PROGRAM Stn6
VAR

	start6: BOOL;
	reset6: BOOL;

	Stn6ProcessFE: F_TRIG;
	Stn6ProcessRE: R_TRIG;
	bCutStn6ProcessHalt: BOOL;
	DoorClose6: R_TRIG;
	bStn6DoorClamp: BOOL;

END_VAR
VAR // added by the converter: edge detectors and wires of the graphical bodies
    _w1, _w2 : ANY;
    _w3 : BOOL;
END_VAR

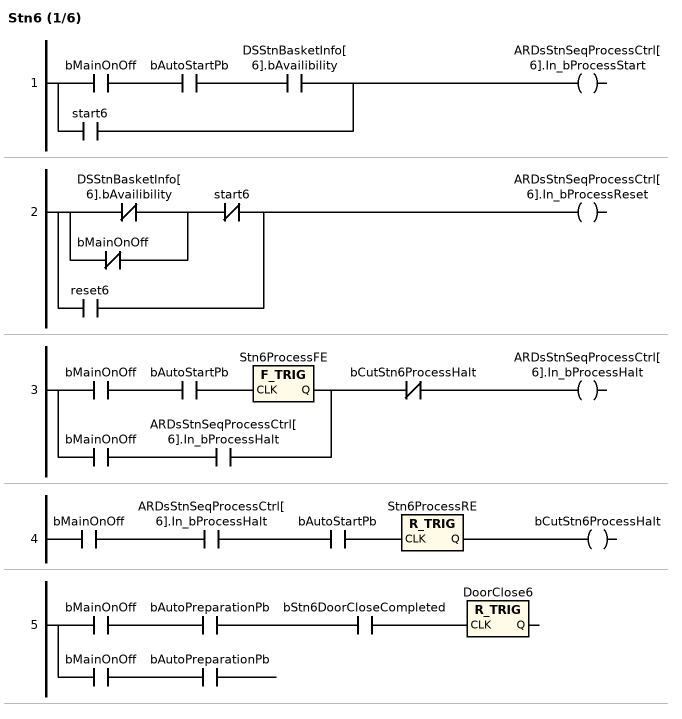
// NETWORK 1
ARDsStnSeqProcessCtrl[6].In_bProcessStart := bMainOnOff AND bAutoStartPb AND DSStnBasketInfo[6].bAvailibility OR start6;

// NETWORK 2
ARDsStnSeqProcessCtrl[6].In_bProcessReset := (NOT DSStnBasketInfo[6].bAvailibility OR NOT bMainOnOff) AND NOT start6 OR reset6;

// NETWORK 3
Stn6ProcessFE(CLK := bMainOnOff AND bAutoStartPb); // F_TRIG
ARDsStnSeqProcessCtrl[6].In_bProcessHalt := (Stn6ProcessFE.Q OR bMainOnOff AND ARDsStnSeqProcessCtrl[6].In_bProcessHalt) AND NOT bCutStn6ProcessHalt;

// NETWORK 4
Stn6ProcessRE(CLK := bMainOnOff AND ARDsStnSeqProcessCtrl[6].In_bProcessHalt AND bAutoStartPb); // R_TRIG
bCutStn6ProcessHalt := Stn6ProcessRE.Q;

// NETWORK 5
DoorClose6(CLK := bMainOnOff AND bAutoPreparationPb AND bStn6DoorCloseCompleted); // R_TRIG
(* DoorClose6.Q OR bMainOnOff AND bAutoPreparationPb; result not used *)

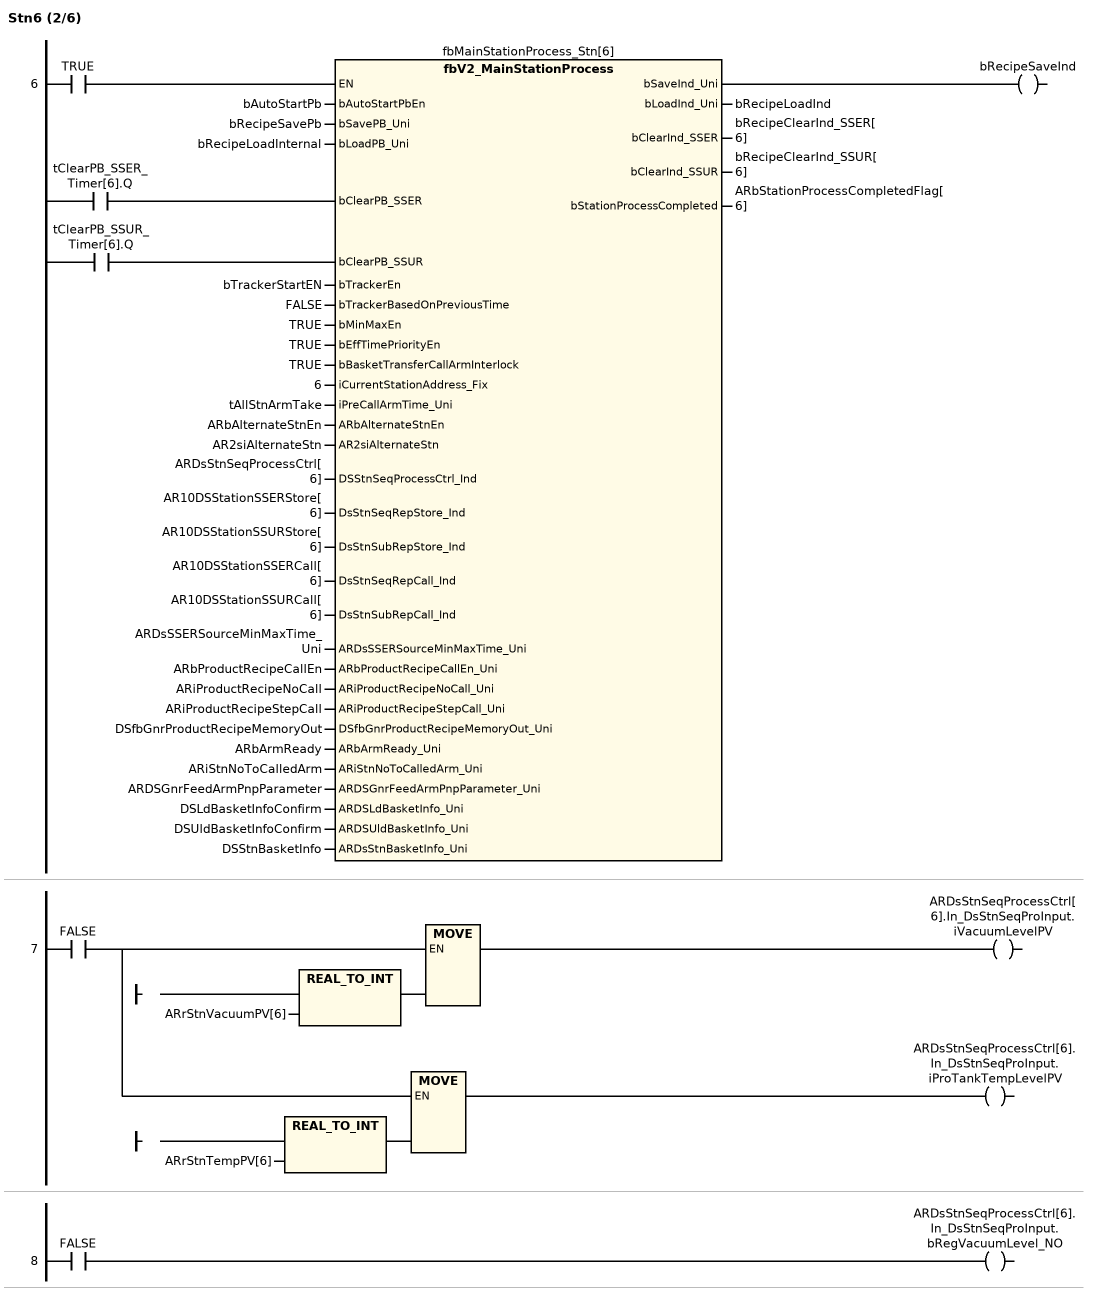
// NETWORK 6
fbMainStationProcess_Stn[6](
    bAutoStartPbEn := bAutoStartPb,
    bSavePB_Uni := bRecipeSavePb,
    bLoadPB_Uni := bRecipeLoadInternal,
    bClearPB_SSER := tClearPB_SSER_Timer[6].Q,
    bClearPB_SSUR := tClearPB_SSUR_Timer[6].Q,
    bTrackerEn := bTrackerStartEN,
    bTrackerBasedOnPreviousTime := FALSE,
    bMinMaxEn := TRUE,
    bEffTimePriorityEn := TRUE,
    bBasketTransferCallArmInterlock := TRUE,
    iCurrentStationAddress_Fix := 6,
    iPreCallArmTime_Uni := tAllStnArmTake,
    ARbAlternateStnEn := ARbAlternateStnEn,
    AR2siAlternateStn := AR2siAlternateStn,
    DSStnSeqProcessCtrl_Ind := ARDsStnSeqProcessCtrl[6],
    DsStnSeqRepStore_Ind := AR10DSStationSSERStore[6],
    DsStnSubRepStore_Ind := AR10DSStationSSURStore[6],
    DsStnSeqRepCall_Ind := AR10DSStationSSERCall[6],
    DsStnSubRepCall_Ind := AR10DSStationSSURCall[6],
    ARDsSSERSourceMinMaxTime_Uni := ARDsSSERSourceMinMaxTime_Uni,
    ARbProductRecipeCallEn_Uni := ARbProductRecipeCallEn,
    ARiProductRecipeNoCall_Uni := ARiProductRecipeNoCall,
    ARiProductRecipeStepCall_Uni := ARiProductRecipeStepCall,
    DSfbGnrProductRecipeMemoryOut_Uni := DSfbGnrProductRecipeMemoryOut,
    ARbArmReady_Uni := ARbArmReady,
    ARiStnNoToCalledArm_Uni := ARiStnNoToCalledArm,
    ARDSGnrFeedArmPnpParameter_Uni := ARDSGnrFeedArmPnpParameter,
    ARDSLdBasketInfo_Uni := DSLdBasketInfoConfirm,
    ARDSUldBasketInfo_Uni := DSUldBasketInfoConfirm,
    ARDsStnBasketInfo_Uni := DSStnBasketInfo,
    bLoadInd_Uni => bRecipeLoadInd,
    bClearInd_SSER => bRecipeClearInd_SSER[6],
    bClearInd_SSUR => bRecipeClearInd_SSUR[6],
    bStationProcessCompleted => ARbStationProcessCompletedFlag[6]); // fbV2_MainStationProcess
bRecipeSaveInd := fbMainStationProcess_Stn[6].bSaveInd_Uni;

// NETWORK 7
IF FALSE THEN _w1 := REAL_TO_INT(ARrStnVacuumPV[6]); END_IF
ARDsStnSeqProcessCtrl[6].In_DsStnSeqProInput.iVacuumLevelPV := _w1;
IF FALSE THEN _w2 := REAL_TO_INT(ARrStnTempPV[6]); END_IF
ARDsStnSeqProcessCtrl[6].In_DsStnSeqProInput.iProTankTempLevelPV := _w2;

// NETWORK 8
ARDsStnSeqProcessCtrl[6].In_DsStnSeqProInput.bRegVacuumLevel_NO := FALSE;

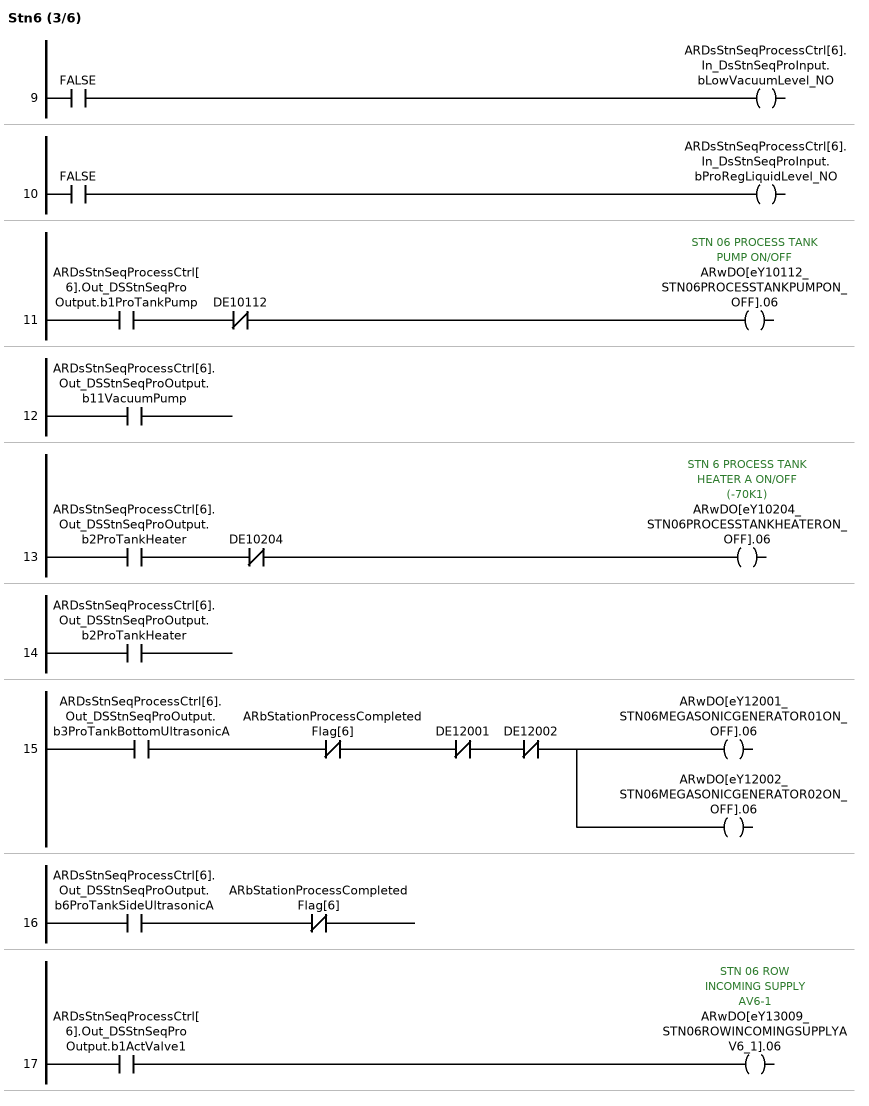
// NETWORK 9
ARDsStnSeqProcessCtrl[6].In_DsStnSeqProInput.bLowVacuumLevel_NO := FALSE;

// NETWORK 10
ARDsStnSeqProcessCtrl[6].In_DsStnSeqProInput.bProRegLiquidLevel_NO := FALSE;

// NETWORK 11
//   ARwDO[eY10112_STN06PROCESSTANKPUMPON_OFF].06: STN 06 PROCESS TANK PUMP ON/OFF
ARwDO[eY10112_STN06PROCESSTANKPUMPON_OFF].06 := ARDsStnSeqProcessCtrl[6].Out_DSStnSeqProOutput.b1ProTankPump AND NOT DE10112;

// NETWORK 12
(* ARDsStnSeqProcessCtrl[6].Out_DSStnSeqProOutput.b11VacuumPump; not connected *)

// NETWORK 13
//   ARwDO[eY10204_STN06PROCESSTANKHEATERON_OFF].06: STN 6 PROCESS TANK HEATER A ON/OFF (-70K1)
ARwDO[eY10204_STN06PROCESSTANKHEATERON_OFF].06 := ARDsStnSeqProcessCtrl[6].Out_DSStnSeqProOutput.b2ProTankHeater AND NOT DE10204;

// NETWORK 14
(* ARDsStnSeqProcessCtrl[6].Out_DSStnSeqProOutput.b2ProTankHeater; not connected *)

// NETWORK 15
_w3 := ARDsStnSeqProcessCtrl[6].Out_DSStnSeqProOutput.b3ProTankBottomUltrasonicA AND NOT ARbStationProcessCompletedFlag[6] AND NOT DE12001 AND NOT DE12002;
ARwDO[eY12001_STN06MEGASONICGENERATOR01ON_OFF].06 := _w3;
ARwDO[eY12002_STN06MEGASONICGENERATOR02ON_OFF].06 := _w3;

// NETWORK 16
(* ARDsStnSeqProcessCtrl[6].Out_DSStnSeqProOutput.b6ProTankSideUltrasonicA AND NOT ARbStationProcessCompletedFlag[6]; result not used *)

// NETWORK 17
//   ARwDO[eY13009_STN06ROWINCOMINGSUPPLYAV6_1].06: STN 06 ROW INCOMING SUPPLY AV6-1
ARwDO[eY13009_STN06ROWINCOMINGSUPPLYAV6_1].06 := ARDsStnSeqProcessCtrl[6].Out_DSStnSeqProOutput.b1ActValve1;

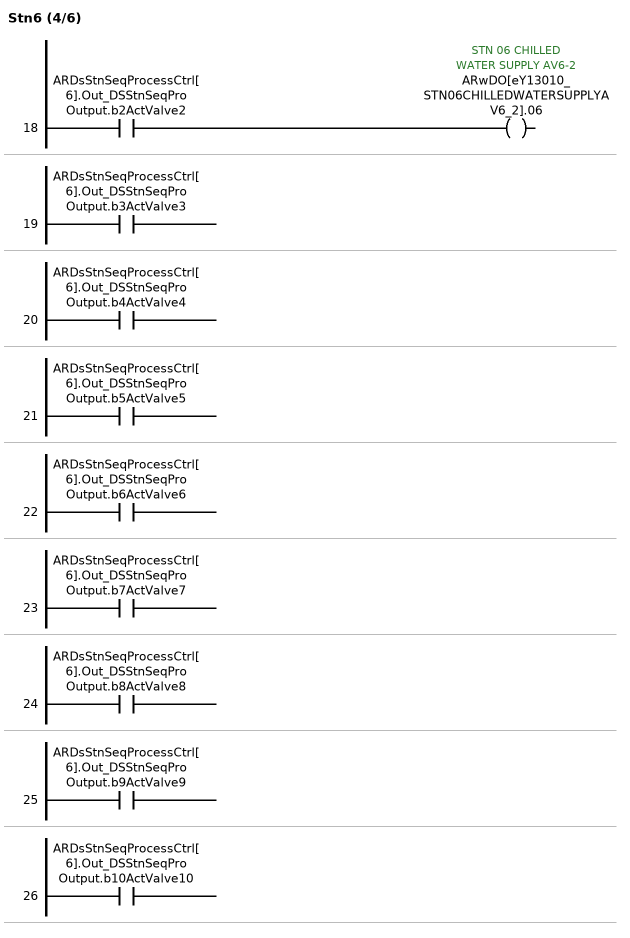
// NETWORK 18
//   ARwDO[eY13010_STN06CHILLEDWATERSUPPLYAV6_2].06: STN 06 CHILLED WATER SUPPLY AV6-2
ARwDO[eY13010_STN06CHILLEDWATERSUPPLYAV6_2].06 := ARDsStnSeqProcessCtrl[6].Out_DSStnSeqProOutput.b2ActValve2;

// NETWORK 19
(* ARDsStnSeqProcessCtrl[6].Out_DSStnSeqProOutput.b3ActValve3; not connected *)

// NETWORK 20
(* ARDsStnSeqProcessCtrl[6].Out_DSStnSeqProOutput.b4ActValve4; not connected *)

// NETWORK 21
(* ARDsStnSeqProcessCtrl[6].Out_DSStnSeqProOutput.b5ActValve5; not connected *)

// NETWORK 22
(* ARDsStnSeqProcessCtrl[6].Out_DSStnSeqProOutput.b6ActValve6; not connected *)

// NETWORK 23
(* ARDsStnSeqProcessCtrl[6].Out_DSStnSeqProOutput.b7ActValve7; not connected *)

// NETWORK 24
(* ARDsStnSeqProcessCtrl[6].Out_DSStnSeqProOutput.b8ActValve8; not connected *)

// NETWORK 25
(* ARDsStnSeqProcessCtrl[6].Out_DSStnSeqProOutput.b9ActValve9; not connected *)

// NETWORK 26
(* ARDsStnSeqProcessCtrl[6].Out_DSStnSeqProOutput.b10ActValve10; not connected *)

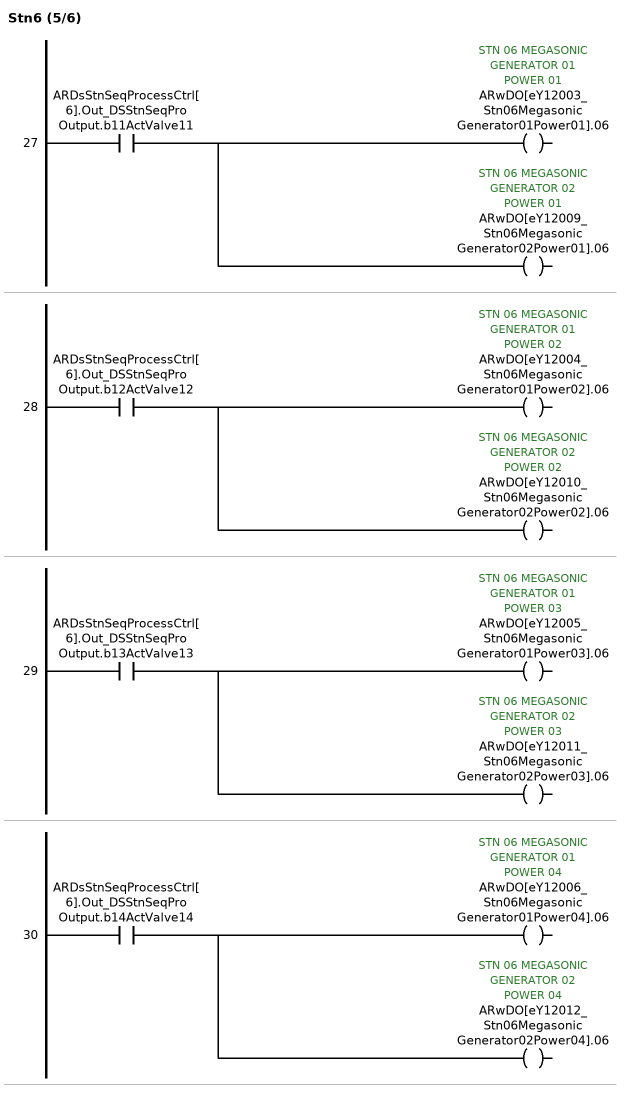
// NETWORK 27
//   ARwDO[eY12003_Stn06MegasonicGenerator01Power01].06: STN 06 MEGASONIC GENERATOR 01 POWER 01
//   ARwDO[eY12009_Stn06MegasonicGenerator02Power01].06: STN 06 MEGASONIC GENERATOR 02 POWER 01
ARwDO[eY12003_Stn06MegasonicGenerator01Power01].06 := ARDsStnSeqProcessCtrl[6].Out_DSStnSeqProOutput.b11ActValve11;
ARwDO[eY12009_Stn06MegasonicGenerator02Power01].06 := ARDsStnSeqProcessCtrl[6].Out_DSStnSeqProOutput.b11ActValve11;

// NETWORK 28
//   ARwDO[eY12004_Stn06MegasonicGenerator01Power02].06: STN 06 MEGASONIC GENERATOR 01 POWER 02
//   ARwDO[eY12010_Stn06MegasonicGenerator02Power02].06: STN 06 MEGASONIC GENERATOR 02 POWER 02
ARwDO[eY12004_Stn06MegasonicGenerator01Power02].06 := ARDsStnSeqProcessCtrl[6].Out_DSStnSeqProOutput.b12ActValve12;
ARwDO[eY12010_Stn06MegasonicGenerator02Power02].06 := ARDsStnSeqProcessCtrl[6].Out_DSStnSeqProOutput.b12ActValve12;

// NETWORK 29
//   ARwDO[eY12005_Stn06MegasonicGenerator01Power03].06: STN 06 MEGASONIC GENERATOR 01 POWER 03
//   ARwDO[eY12011_Stn06MegasonicGenerator02Power03].06: STN 06 MEGASONIC GENERATOR 02 POWER 03
ARwDO[eY12005_Stn06MegasonicGenerator01Power03].06 := ARDsStnSeqProcessCtrl[6].Out_DSStnSeqProOutput.b13ActValve13;
ARwDO[eY12011_Stn06MegasonicGenerator02Power03].06 := ARDsStnSeqProcessCtrl[6].Out_DSStnSeqProOutput.b13ActValve13;

// NETWORK 30
//   ARwDO[eY12006_Stn06MegasonicGenerator01Power04].06: STN 06 MEGASONIC GENERATOR 01 POWER 04
//   ARwDO[eY12012_Stn06MegasonicGenerator02Power04].06: STN 06 MEGASONIC GENERATOR 02 POWER 04
ARwDO[eY12006_Stn06MegasonicGenerator01Power04].06 := ARDsStnSeqProcessCtrl[6].Out_DSStnSeqProOutput.b14ActValve14;
ARwDO[eY12012_Stn06MegasonicGenerator02Power04].06 := ARDsStnSeqProcessCtrl[6].Out_DSStnSeqProOutput.b14ActValve14;

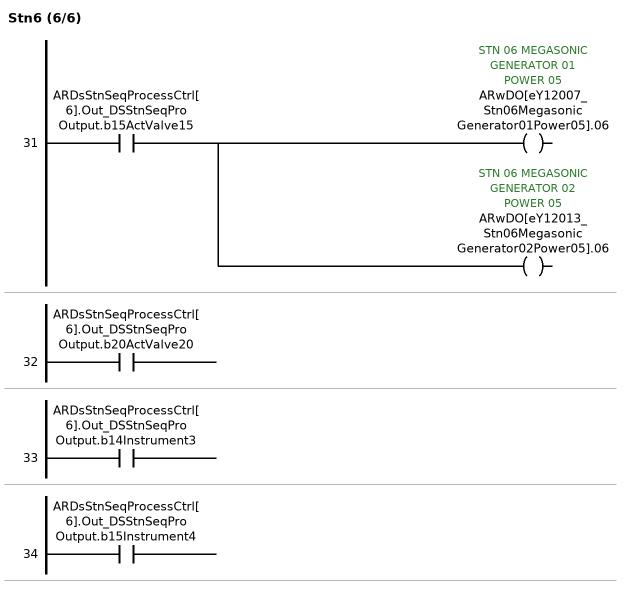
// NETWORK 31
//   ARwDO[eY12007_Stn06MegasonicGenerator01Power05].06: STN 06 MEGASONIC GENERATOR 01 POWER 05
//   ARwDO[eY12013_Stn06MegasonicGenerator02Power05].06: STN 06 MEGASONIC GENERATOR 02 POWER 05
ARwDO[eY12007_Stn06MegasonicGenerator01Power05].06 := ARDsStnSeqProcessCtrl[6].Out_DSStnSeqProOutput.b15ActValve15;
ARwDO[eY12013_Stn06MegasonicGenerator02Power05].06 := ARDsStnSeqProcessCtrl[6].Out_DSStnSeqProOutput.b15ActValve15;

// NETWORK 32
(* ARDsStnSeqProcessCtrl[6].Out_DSStnSeqProOutput.b20ActValve20; not connected *)

// NETWORK 33
(* ARDsStnSeqProcessCtrl[6].Out_DSStnSeqProOutput.b14Instrument3; not connected *)

// NETWORK 34
(* ARDsStnSeqProcessCtrl[6].Out_DSStnSeqProOutput.b15Instrument4; not connected *)

END_PROGRAM

(* stored: Version 1.1.0.1, ProductVersion 3.1.4024.12
   POU Stn6: Id {39a51eaf-bbaf-4fdd-aa32-b0cb7a1e6c08}, SpecialFunc None *)
